// Brief: Slave Arm Run Self-check Trajectory
FUNCTION_BLOCK PUBLIC FB_SlaveCtrlSelfCheck EXTENDS FB_SlaveArmCtrlBase

VAR
	// slave self-check motion parameters
	m_selfCheckPosture:ARRAY [1..g_sJntNum] OF LREAL:=[0.0,	-PI/2,	GVL_SlaveMotorParameters.g_maxDHJntPos[3], 	5(-g_2pi)];																			//PI/4, -PI/4, 0.3, pi, pi, pi, pi, pi];
	m_selfCheckMaxjntVel:Vec8d:=[2(20*g_deg2Rad),  0.3/2, 5(2*pi)];
	m_selfCheckMaxjntAcc:Vec8d:=[2(20*g_deg2Rad), 	0.6/2, 5(4*pi)];
	m_selfCheckMaxjntJerk:Vec8d:=[2(20*g_deg2Rad),  1.0/2, 5(8*pi)];
	
	m_slefCheckPlanner: ARRAY[1..g_sJntNum] OF FB_BasicDoubleS;
	
   // wait time for joint enable
   m_enableWaitTime :LREAL := 1.0;

   // time wait to motion
   m_jntMotionWaitTime :LREAL := 3.0;
   
   m_selfCheckMotionKp :LREAL := 10;
   m_jntVelFilt :ARRAY[1..2] OF FB_LowPassFilter;

END_VAR

// override this function in each exact controller
METHOD PROTECTED calcCmdJntPos : BOOL
VAR_IN_OUT CONSTANT
	i_endoscopePose : ST_Frame;
	i_masterStatus :ST_MasterStatus;
	i_setupStatus: ST_SetupStatus;
	i_slaveArm :FB_SlaveArm;
END_VAR

VAR 
	i :INT;
	curJntPos :Vec8d;
	posErr:Vec8d;
END_VAR
// check if planner is ready
FOR i:=3 TO g_sJntNum DO 
	IF m_slefCheckPlanner[i].isGene = FALSE THEN
		calcCmdJntPos:=FALSE;
		RETURN;
	END_IF
END_FOR  

// arms enable successively
IF m_timePeriod > m_enableWaitTime THEN
       m_jntEnableFlag :=g_onesVec8i;
END_IF

IF m_timePeriod < m_jntMotionWaitTime THEN
	RETURN;
END_IF

// traj plan
FOR i:=3 TO g_sJntNum DO 
	calcCmdJntPos :=m_slefCheckPlanner[i].evaluate(m_timePeriod-m_jntMotionWaitTime, q=> m_cmdJntPos[i], q_dot=>m_cmdJntVel[i], q_ddot=> m_cmdJntAcc[i]);
END_FOR 

// self-collision avoid motion 
FOR i:=1 TO 2 DO 
	m_cmdJntVel[i] := m_selfCheckMotionKp *(m_selfCheckPosture[i]-m_cmdJntPos[i]);
	m_cmdJntVel[i] := LIMIT(-m_selfCheckMaxjntVel[i], m_cmdJntVel[i], m_selfCheckMaxjntVel[i]);
	m_cmdJntVel[i]:=m_jntVelFilt[i].run(m_cmdJntVel[i]+i_slaveArm.m_repulseJntVel[i]);
	
	// boundary limit
	IF (m_cmdJntPos[i] > GVL_SlaveMotorParameters.g_maxDHJntPos[i] AND m_cmdJntVel[i] > 0) OR
		(m_cmdJntPos[i] < GVL_SlaveMotorParameters.g_minDHJntPos[i] AND m_cmdJntVel[i] < 0) THEN
		m_cmdJntVel[i] :=0;
	END_IF
	
	m_cmdJntPos[i] := m_cmdJntPos[i] + m_cmdJntVel[i] * g_slaveArmCtrlCycleTime;
END_FOR

// check if to terminated
curJntPos := i_slaveArm.curJntPos;
vecSub(m_selfCheckPosture, curJntPos, posErr);
m_isFinished := TRUE;
FOR i:=1 TO g_sJntNum DO
	IF (i=3 AND ABS(posErr[i]) > g_cartCtrlPosTolHigh/2.0) OR (i<>3 AND ABS(posErr[i]) > g_jntCtrlAngTolHigh/2.0) THEN
		m_isFinished := FALSE;
		RETURN;
	END_IF
END_FOR
END_METHOD

METHOD PUBLIC init : BOOL
VAR_IN_OUT CONSTANT
	i_slaveArm	:FB_SlaveArm;
END_VAR
VAR_IN_OUT 
	r_slaveArmCtrlCmd :ST_SlaveArmCtrlCmds;
END_VAR

VAR_STAT
	i :INT;
	baseJntPos:Vec8d;
	cycleNum :LREAL;
	q,v :Vec2d;
END_VAR
SUPER^.Init(i_slaveArm,r_slaveArmCtrlCmd);
m_jntEnableFlag :=g_zeroVec8i;

//set different wait time for each arm, so the arms would run self-check successively
m_enableWaitTime := (i_slaveArm.armIdx-1.0)/2.0;
m_selfCheckPosture[3] := GVL_SlaveMotorParameters.g_maxDHJntPos[3];

// determine base joint position for instrument joint
baseJntPos :=g_zeroVec8d;
FOR i:=4 TO g_sJntNum DO
		cycleNum := FLOOR(i_slaveArm.curJntPos[i]/(2*pi));
		baseJntPos[i]:=cycleNum* g_2Pi;
		m_selfCheckPosture[i]:=baseJntPos[i] + m_selfCheckPosture[i];
END_FOR

// traj plan for joint 3-8
FOR i:=3 TO g_sJntNum DO 
	q[1]:=i_slaveArm.curJntPos[i];
	q[2]:=m_selfCheckPosture[i];
	v[1]:=0;
	v[2]:=0;
	m_slefCheckPlanner[i].init(q,v,m_selfCheckMaxjntVel[i], m_selfCheckMaxjntAcc[i], m_selfCheckMaxjntJerk[i]);
END_FOR

FOR i:=1 TO 2 DO
	m_jntVelFilt[i].init(1, 1, g_slaveArmCtrlFreq);
	m_jntVelFilt[i].run(0);;
END_FOR

//check trocar on
IF CartControl.m_cartRobot.m_slaveCart.m_trocarOnFlag > 0 THEN
	m_selfCheckPosture[1]:=i_slaveArm.curJntPos[1];
	m_selfCheckPosture[2]:=i_slaveArm.curJntPos[2];
END_IF

// update commands to arm
copyCmds(r_slaveArmCtrlCmd);
END_METHOD

END_FUNCTION_BLOCK

(* stored: Version 1.1.0.1, ProductVersion 3.1.4024.11
   POU FB_SlaveCtrlSelfCheck: Id {ff8ccb3f-4929-4315-b540-e9546f2dbd07}, SpecialFunc None
   Method calcCmdJntPos: Id {ffa3dbdd-63a1-4101-8d26-d1f3e6e5e2be}
   Method init: Id {c6523e12-84cb-49f8-843e-9a168bb4ce28} *)
